INTERFACE I_FallibleSTRING EXTENDS I_Fallible

PROPERTY Val : STRING
GET
END_GET
END_PROPERTY

END_INTERFACE

(* stored: Version 1.1.0.1
   Itf I_FallibleSTRING: Id {2957f111-c4c0-4ae9-afb9-8752f870f9b8}
   Property Val: Id {ef08e5ad-69a5-45ca-90a0-91991e28fbfe}
   Get Get: Id {bdb08467-f5ea-4405-88bc-28b848ed4b8c} *)
